TYPE ST_TsDiagObjectsEL1904 :
(*******************************************************************************************************
Description			:	Index 16#800E Diagnostic objects
Supported terminals : 	EL1904
********************************************************************************************************)
STRUCT

	nNotUsedData1								:ARRAY[0..8] OF UINT;

(* Sensor test error *)
	nSensorTestError						:UINT;
	(*TsDiagObjectsBitsEL1904_bSensorTestError_Input1		 		:= stDiagObjects.nSensorTestError.0;
	TsDiagObjectsBitsEL1904_bSensorTestError_Input2		 			 := stDiagObjects.nSensorTestError.1;
	TsDiagObjectsBitsEL1904_bSensorTestError_Input3		 			 := stDiagObjects.nSensorTestError.2;
	TsDiagObjectsBitsEL1904_bSensorTestError_Input4		 			 := stDiagObjects.nSensorTestError.3;*)
	

(* Error during two channel evaluation *)
	nDuringTwoChannelEvaluationError		:UINT;
	(*TsDiagObjectsBitsEL1904_bErrFirstInputPair 			 := stDiagObjects.nDuringTwoChannelEvaluationError.0;
	TsDiagObjectsBitsEL1904_bErrSecondInputPair 		 := stDiagObjects.nDuringTwoChannelEvaluationError.1;*)


(* Error in the safety mat operating mode: input pair disagree *)
	nMatModeInputPairDisagreeError			:UINT;
	(*TsDiagObjectsBitsEL1904_bMatOpModeErrFirstInputPair	 := stDiagObjects.nMatModeInputPairDisagreeError.0 
																			AND stDiagObjects.nMatModeInputPairDisagreeError.1;
	TsDiagObjectsBitsEL1904_bMatOpModeErrSecondInputPair := stDiagObjects.nMatModeInputPairDisagreeError.2 
																			AND stDiagObjects.nMatModeInputPairDisagreeError.3;*)
	
(* Error in the safety mat operating mode: external supply *)
	nMatModeExternalSupplyError				:UINT;
	(*TsDiagObjectsBitsEL1904_bMatOpModeExtSupplyError_Input1 := stDiagObjects.nMatModeExternalSupplyError.0;
	TsDiagObjectsBitsEL1904_bMatOpModeExtSupplyError_Input2 := stDiagObjects.nMatModeExternalSupplyError.1;
	TsDiagObjectsBitsEL1904_bMatOpModeExtSupplyError_Input3 := stDiagObjects.nMatModeExternalSupplyError.2;
	TsDiagObjectsBitsEL1904_bMatOpModeExtSupplyError_Input4 := stDiagObjects.nMatModeExternalSupplyError.3;*)
	
	nNotUsedData2								:ARRAY[0..2] OF UINT;

END_STRUCT
END_TYPE
(* End *)

(* stored: Version 1.1.0.1, ProductVersion 3.1.4024.12
   DUT ST_TsDiagObjectsEL1904: Id {911e5244-c753-4991-9599-f9d8ff4e3592} *)
